# B&R Automation Studio project BaR_Automation_Studio
Automation Studio 4.9

## Configuration Config_5APC2100

CPU 5APC2100.BY48-000, AutomationRuntime B4.83, Build 4.1.2, Safety 1.10, Vc V4.72.6

### IoMap.iom - 5APC2100_BY48_000/IoMap.iom
```iecst
VAR_CONFIG
	::RESET_SAFETY AT %QX."X20SLX842".BOOL101;
	::Global_VInRoS_Str.EX_600.Slave.Info.Active AT %IX."EX600_WEN__V1_1".ModuleOk;
	::T_EX600:C_USINT_To_BOOL_Arr_1.INPUT AT %IB."EX600_WEN__V1_1".Module_0_Input011;
	::T_EX600:C_USINT_To_BOOL_Arr_2.INPUT AT %IB."EX600_WEN__V1_1".Module_0_Input012;
	::T_EX600:C_BOOL_Arr_To_USINT_1.OUTPUT AT %QB."EX600_WEN__V1_1".Module_0_Output003;
	::SAFETY_ACTIVE AT %IX."X20SLX842".SafeDigitalInput03;
	::SAFETY_STATUS AT %IX."X20SLX842".BOOL001;
	::T_ROB_1:ABB_Library_Rob_1.Status.PLC.Module_OK AT %IX."BASIC_V1_2".ModuleOk;
	::T_ROB_1:ABB_Library_Rob_1.PROFINET_Mapping_IN.STATUS.INPUT AT %IB."BASIC_V1_2".Module001_Input_0;
	::T_ROB_1:ABB_Library_Rob_1.PROFINET_Mapping_IN.SYSTEM.INPUT AT %IB."BASIC_V1_2".Module001_Input_1;
	::T_ROB_1:ABB_Library_Rob_1.PROFINET_Mapping_IN.STATE_uID AT %IB."BASIC_V1_2".Module001_Input_2;
	::T_ROB_1:ABB_Library_Rob_1.PROFINET_Mapping_IN.STATE_mID AT %IB."BASIC_V1_2".Module001_Input_3;
	::T_ROB_1:ABB_Library_Rob_1.PROFINET_Mapping_IN.MOTION_TRAJECTORY_ID.INPUT[0] AT %IB."BASIC_V1_2".Module001_Input_4;
	::T_ROB_1:ABB_Library_Rob_1.PROFINET_Mapping_IN.MOTION_TRAJECTORY_ID.INPUT[1] AT %IB."BASIC_V1_2".Module001_Input_5;
	::T_ROB_1:ABB_Library_Rob_1.PROFINET_Mapping_IN.JOINT_POS[0].INPUT[0] AT %IB."BASIC_V1_2".Module001_Input_6;
	::T_ROB_1:ABB_Library_Rob_1.PROFINET_Mapping_IN.JOINT_POS[0].INPUT[1] AT %IB."BASIC_V1_2".Module001_Input_7;
	::T_ROB_1:ABB_Library_Rob_1.PROFINET_Mapping_IN.JOINT_POS[1].INPUT[0] AT %IB."BASIC_V1_2".Module001_Input_8;
	::T_ROB_1:ABB_Library_Rob_1.PROFINET_Mapping_IN.JOINT_POS[1].INPUT[1] AT %IB."BASIC_V1_2".Module001_Input_9;
	::T_ROB_1:ABB_Library_Rob_1.PROFINET_Mapping_IN.JOINT_POS[2].INPUT[0] AT %IB."BASIC_V1_2".Module001_Input_10;
	::T_ROB_1:ABB_Library_Rob_1.PROFINET_Mapping_IN.JOINT_POS[2].INPUT[1] AT %IB."BASIC_V1_2".Module001_Input_11;
	::T_ROB_1:ABB_Library_Rob_1.PROFINET_Mapping_IN.JOINT_POS[3].INPUT[0] AT %IB."BASIC_V1_2".Module001_Input_12;
	::T_ROB_1:ABB_Library_Rob_1.PROFINET_Mapping_IN.JOINT_POS[3].INPUT[1] AT %IB."BASIC_V1_2".Module001_Input_13;
	::T_ROB_1:ABB_Library_Rob_1.PROFINET_Mapping_IN.JOINT_POS[4].INPUT[0] AT %IB."BASIC_V1_2".Module001_Input_14;
	::T_ROB_1:ABB_Library_Rob_1.PROFINET_Mapping_IN.JOINT_POS[4].INPUT[1] AT %IB."BASIC_V1_2".Module001_Input_15;
	::T_ROB_1:ABB_Library_Rob_1.PROFINET_Mapping_IN.JOINT_POS[5].INPUT[0] AT %IB."BASIC_V1_2".Module001_Input_16;
	::T_ROB_1:ABB_Library_Rob_1.PROFINET_Mapping_IN.JOINT_POS[5].INPUT[1] AT %IB."BASIC_V1_2".Module001_Input_17;
	::T_ROB_1:ABB_Library_Rob_1.PROFINET_Mapping_IN.JOINT_POS[6].INPUT[0] AT %IB."BASIC_V1_2".Module001_Input_18;
	::T_ROB_1:ABB_Library_Rob_1.PROFINET_Mapping_IN.JOINT_POS[6].INPUT[1] AT %IB."BASIC_V1_2".Module001_Input_19;
	::T_ROB_1:ABB_Library_Rob_1.PROFINET_Mapping_IN.JOINT_POS_SIGN.INPUT AT %IB."BASIC_V1_2".Module001_Input_20;
	::T_ROB_1:ABB_Library_Rob_1.PROFINET_Mapping_IN.TCP_POS[0].INPUT[0] AT %IB."BASIC_V1_2".Module001_Input_21;
	::T_ROB_1:ABB_Library_Rob_1.PROFINET_Mapping_IN.TCP_POS[0].INPUT[1] AT %IB."BASIC_V1_2".Module001_Input_22;
	::T_ROB_1:ABB_Library_Rob_1.PROFINET_Mapping_IN.TCP_POS[0].INPUT[2] AT %IB."BASIC_V1_2".Module001_Input_23;
	::T_ROB_1:ABB_Library_Rob_1.PROFINET_Mapping_IN.TCP_POS[0].INPUT[3] AT %IB."BASIC_V1_2".Module001_Input_24;
	::T_ROB_1:ABB_Library_Rob_1.PROFINET_Mapping_IN.TCP_POS[1].INPUT[0] AT %IB."BASIC_V1_2".Module001_Input_25;
	::T_ROB_1:ABB_Library_Rob_1.PROFINET_Mapping_IN.TCP_POS[1].INPUT[1] AT %IB."BASIC_V1_2".Module001_Input_26;
	::T_ROB_1:ABB_Library_Rob_1.PROFINET_Mapping_IN.TCP_POS[1].INPUT[2] AT %IB."BASIC_V1_2".Module001_Input_27;
	::T_ROB_1:ABB_Library_Rob_1.PROFINET_Mapping_IN.TCP_POS[1].INPUT[3] AT %IB."BASIC_V1_2".Module001_Input_28;
	::T_ROB_1:ABB_Library_Rob_1.PROFINET_Mapping_IN.TCP_POS[2].INPUT[0] AT %IB."BASIC_V1_2".Module001_Input_29;
	::T_ROB_1:ABB_Library_Rob_1.PROFINET_Mapping_IN.TCP_POS[2].INPUT[1] AT %IB."BASIC_V1_2".Module001_Input_30;
	::T_ROB_1:ABB_Library_Rob_1.PROFINET_Mapping_IN.TCP_POS[2].INPUT[2] AT %IB."BASIC_V1_2".Module001_Input_31;
	::T_ROB_1:ABB_Library_Rob_1.PROFINET_Mapping_IN.TCP_POS[2].INPUT[3] AT %IB."BASIC_V1_2".Module001_Input_32;
	::T_ROB_1:ABB_Library_Rob_1.PROFINET_Mapping_IN.TCP_ROT[0].INPUT[0] AT %IB."BASIC_V1_2".Module001_Input_33;
	::T_ROB_1:ABB_Library_Rob_1.PROFINET_Mapping_IN.TCP_ROT[0].INPUT[1] AT %IB."BASIC_V1_2".Module001_Input_34;
	::T_ROB_1:ABB_Library_Rob_1.PROFINET_Mapping_IN.TCP_ROT[1].INPUT[0] AT %IB."BASIC_V1_2".Module001_Input_35;
	::T_ROB_1:ABB_Library_Rob_1.PROFINET_Mapping_IN.TCP_ROT[1].INPUT[1] AT %IB."BASIC_V1_2".Module001_Input_36;
	::T_ROB_1:ABB_Library_Rob_1.PROFINET_Mapping_IN.TCP_ROT[2].INPUT[0] AT %IB."BASIC_V1_2".Module001_Input_37;
	::T_ROB_1:ABB_Library_Rob_1.PROFINET_Mapping_IN.TCP_ROT[2].INPUT[1] AT %IB."BASIC_V1_2".Module001_Input_38;
	::T_ROB_1:ABB_Library_Rob_1.PROFINET_Mapping_IN.TCP_EX_POS.INPUT[0] AT %IB."BASIC_V1_2".Module001_Input_39;
	::T_ROB_1:ABB_Library_Rob_1.PROFINET_Mapping_IN.TCP_EX_POS.INPUT[1] AT %IB."BASIC_V1_2".Module001_Input_40;
	::T_ROB_1:ABB_Library_Rob_1.PROFINET_Mapping_IN.TCP_SIGN.INPUT AT %IB."BASIC_V1_2".Module001_Input_41;
	::T_ROB_1:ABB_Library_Rob_1.PROFINET_Mapping_IN.TCP_CFG[0] AT %IB."BASIC_V1_2".Module001_Input_42;
	::T_ROB_1:ABB_Library_Rob_1.PROFINET_Mapping_IN.TCP_CFG[1] AT %IB."BASIC_V1_2".Module001_Input_43;
	::T_ROB_1:ABB_Library_Rob_1.PROFINET_Mapping_IN.TCP_CFG[2] AT %IB."BASIC_V1_2".Module001_Input_44;
	::T_ROB_1:ABB_Library_Rob_1.PROFINET_Mapping_IN.TCP_CFG[3] AT %IB."BASIC_V1_2".Module001_Input_45;
	::T_ROB_1:ABB_Library_Rob_1.PROFINET_Mapping_IN.TCP_CFG_SIGN.INPUT AT %IB."BASIC_V1_2".Module001_Input_46;
	::T_ROB_1:ABB_Library_Rob_1.PROFINET_Mapping_OUT.STATUS.OUTPUT AT %QB."BASIC_V1_2".Module002_Output_0;
	::T_ROB_1:ABB_Library_Rob_1.PROFINET_Mapping_OUT.SYSTEM.OUTPUT AT %QB."BASIC_V1_2".Module002_Output_1;
	::T_ROB_1:ABB_Library_Rob_1.PROFINET_Mapping_OUT.COMMAND.OUTPUT AT %QB."BASIC_V1_2".Module002_Output_2;
	::T_ROB_1:ABB_Library_Rob_1.PROFINET_Mapping_OUT.COMMAND_mID AT %QB."BASIC_V1_2".Module002_Output_3;
	::T_ROB_1:ABB_Library_Rob_1.PROFINET_Mapping_OUT.COMMAND_uID AT %QB."BASIC_V1_2".Module002_Output_4;
	::T_ROB_1:ABB_Library_Rob_1.PROFINET_Mapping_OUT.TRAJECTORY_SIZE.OUTPUT[0] AT %QB."BASIC_V1_2".Module002_Output_5;
	::T_ROB_1:ABB_Library_Rob_1.PROFINET_Mapping_OUT.TRAJECTORY_SIZE.OUTPUT[1] AT %QB."BASIC_V1_2".Module002_Output_6;
	::T_ROB_1:ABB_Library_Rob_1.PROFINET_Mapping_OUT.SPEED AT %QB."BASIC_V1_2".Module002_Output_7;
	::T_ROB_1:ABB_Library_Rob_1.PROFINET_Mapping_OUT.ZONE AT %QB."BASIC_V1_2".Module002_Output_8;
	::T_ROB_1:ABB_Library_Rob_1.PROFINET_Mapping_OUT.JOINT_POS[0].OUTPUT[0] AT %QB."BASIC_V1_2".Module002_Output_9;
	::T_ROB_1:ABB_Library_Rob_1.PROFINET_Mapping_OUT.JOINT_POS[0].OUTPUT[1] AT %QB."BASIC_V1_2".Module002_Output_10;
	::T_ROB_1:ABB_Library_Rob_1.PROFINET_Mapping_OUT.JOINT_POS[1].OUTPUT[0] AT %QB."BASIC_V1_2".Module002_Output_11;
	::T_ROB_1:ABB_Library_Rob_1.PROFINET_Mapping_OUT.JOINT_POS[1].OUTPUT[1] AT %QB."BASIC_V1_2".Module002_Output_12;
	::T_ROB_1:ABB_Library_Rob_1.PROFINET_Mapping_OUT.JOINT_POS[2].OUTPUT[0] AT %QB."BASIC_V1_2".Module002_Output_13;
	::T_ROB_1:ABB_Library_Rob_1.PROFINET_Mapping_OUT.JOINT_POS[2].OUTPUT[1] AT %QB."BASIC_V1_2".Module002_Output_14;
	::T_ROB_1:ABB_Library_Rob_1.PROFINET_Mapping_OUT.JOINT_POS[3].OUTPUT[0] AT %QB."BASIC_V1_2".Module002_Output_15;
	::T_ROB_1:ABB_Library_Rob_1.PROFINET_Mapping_OUT.JOINT_POS[3].OUTPUT[1] AT %QB."BASIC_V1_2".Module002_Output_16;
	::T_ROB_1:ABB_Library_Rob_1.PROFINET_Mapping_OUT.JOINT_POS[4].OUTPUT[0] AT %QB."BASIC_V1_2".Module002_Output_17;
	::T_ROB_1:ABB_Library_Rob_1.PROFINET_Mapping_OUT.JOINT_POS[4].OUTPUT[1] AT %QB."BASIC_V1_2".Module002_Output_18;
	::T_ROB_1:ABB_Library_Rob_1.PROFINET_Mapping_OUT.JOINT_POS[5].OUTPUT[0] AT %QB."BASIC_V1_2".Module002_Output_19;
	::T_ROB_1:ABB_Library_Rob_1.PROFINET_Mapping_OUT.JOINT_POS[5].OUTPUT[1] AT %QB."BASIC_V1_2".Module002_Output_20;
	::T_ROB_1:ABB_Library_Rob_1.PROFINET_Mapping_OUT.JOINT_POS[6].OUTPUT[0] AT %QB."BASIC_V1_2".Module002_Output_21;
	::T_ROB_1:ABB_Library_Rob_1.PROFINET_Mapping_OUT.JOINT_POS[6].OUTPUT[1] AT %QB."BASIC_V1_2".Module002_Output_22;
	::T_ROB_1:ABB_Library_Rob_1.PROFINET_Mapping_OUT.JOINT_POS_SIGN.OUTPUT AT %QB."BASIC_V1_2".Module002_Output_23;
	::T_ROB_1:ABB_Library_Rob_1.PROFINET_Mapping_OUT.TCP_POS[0].OUTPUT[0] AT %QB."BASIC_V1_2".Module002_Output_24;
	::T_ROB_1:ABB_Library_Rob_1.PROFINET_Mapping_OUT.TCP_POS[0].OUTPUT[1] AT %QB."BASIC_V1_2".Module002_Output_25;
	::T_ROB_1:ABB_Library_Rob_1.PROFINET_Mapping_OUT.TCP_POS[0].OUTPUT[2] AT %QB."BASIC_V1_2".Module002_Output_26;
	::T_ROB_1:ABB_Library_Rob_1.PROFINET_Mapping_OUT.TCP_POS[0].OUTPUT[3] AT %QB."BASIC_V1_2".Module002_Output_27;
	::T_ROB_1:ABB_Library_Rob_1.PROFINET_Mapping_OUT.TCP_POS[1].OUTPUT[0] AT %QB."BASIC_V1_2".Module002_Output_28;
	::T_ROB_1:ABB_Library_Rob_1.PROFINET_Mapping_OUT.TCP_POS[1].OUTPUT[1] AT %QB."BASIC_V1_2".Module002_Output_29;
	::T_ROB_1:ABB_Library_Rob_1.PROFINET_Mapping_OUT.TCP_POS[1].OUTPUT[2] AT %QB."BASIC_V1_2".Module002_Output_30;
	::T_ROB_1:ABB_Library_Rob_1.PROFINET_Mapping_OUT.TCP_POS[1].OUTPUT[3] AT %QB."BASIC_V1_2".Module002_Output_31;
	::T_ROB_1:ABB_Library_Rob_1.PROFINET_Mapping_OUT.TCP_POS[2].OUTPUT[0] AT %QB."BASIC_V1_2".Module002_Output_32;
	::T_ROB_1:ABB_Library_Rob_1.PROFINET_Mapping_OUT.TCP_POS[2].OUTPUT[1] AT %QB."BASIC_V1_2".Module002_Output_33;
	::T_ROB_1:ABB_Library_Rob_1.PROFINET_Mapping_OUT.TCP_POS[2].OUTPUT[2] AT %QB."BASIC_V1_2".Module002_Output_34;
	::T_ROB_1:ABB_Library_Rob_1.PROFINET_Mapping_OUT.TCP_POS[2].OUTPUT[3] AT %QB."BASIC_V1_2".Module002_Output_35;
	::T_ROB_1:ABB_Library_Rob_1.PROFINET_Mapping_OUT.TCP_ROT[0].OUTPUT[0] AT %QB."BASIC_V1_2".Module002_Output_36;
	::T_ROB_1:ABB_Library_Rob_1.PROFINET_Mapping_OUT.TCP_ROT[0].OUTPUT[1] AT %QB."BASIC_V1_2".Module002_Output_37;
	::T_ROB_1:ABB_Library_Rob_1.PROFINET_Mapping_OUT.TCP_ROT[1].OUTPUT[0] AT %QB."BASIC_V1_2".Module002_Output_38;
	::T_ROB_1:ABB_Library_Rob_1.PROFINET_Mapping_OUT.TCP_ROT[1].OUTPUT[1] AT %QB."BASIC_V1_2".Module002_Output_39;
	::T_ROB_1:ABB_Library_Rob_1.PROFINET_Mapping_OUT.TCP_ROT[2].OUTPUT[0] AT %QB."BASIC_V1_2".Module002_Output_40;
	::T_ROB_1:ABB_Library_Rob_1.PROFINET_Mapping_OUT.TCP_ROT[2].OUTPUT[1] AT %QB."BASIC_V1_2".Module002_Output_41;
	::T_ROB_1:ABB_Library_Rob_1.PROFINET_Mapping_OUT.TCP_EX_POS.OUTPUT[0] AT %QB."BASIC_V1_2".Module002_Output_42;
	::T_ROB_1:ABB_Library_Rob_1.PROFINET_Mapping_OUT.TCP_EX_POS.OUTPUT[1] AT %QB."BASIC_V1_2".Module002_Output_43;
	::T_ROB_1:ABB_Library_Rob_1.PROFINET_Mapping_OUT.TCP_SIGN.OUTPUT AT %QB."BASIC_V1_2".Module002_Output_44;
	::T_ROB_1:ABB_Library_Rob_1.PROFINET_Mapping_OUT.TCP_CFG[0] AT %QB."BASIC_V1_2".Module002_Output_45;
	::T_ROB_1:ABB_Library_Rob_1.PROFINET_Mapping_OUT.TCP_CFG[1] AT %QB."BASIC_V1_2".Module002_Output_46;
	::T_ROB_1:ABB_Library_Rob_1.PROFINET_Mapping_OUT.TCP_CFG[2] AT %QB."BASIC_V1_2".Module002_Output_47;
	::T_ROB_1:ABB_Library_Rob_1.PROFINET_Mapping_OUT.TCP_CFG[3] AT %QB."BASIC_V1_2".Module002_Output_48;
	::T_ROB_1:ABB_Library_Rob_1.PROFINET_Mapping_OUT.TCP_CFG_SIGN.OUTPUT AT %QB."BASIC_V1_2".Module002_Output_49;
	::T_ROB_1:ABB_Library_Rob_1.PROFINET_Mapping_OUT.RTOOL_RH.OUTPUT AT %QB."BASIC_V1_2".Module002_Output_50;
	::T_ROB_1:ABB_Library_Rob_1.PROFINET_Mapping_OUT.RTOOL_POS[0].OUTPUT[0] AT %QB."BASIC_V1_2".Module002_Output_51;
	::T_ROB_1:ABB_Library_Rob_1.PROFINET_Mapping_OUT.RTOOL_POS[0].OUTPUT[1] AT %QB."BASIC_V1_2".Module002_Output_52;
	::T_ROB_1:ABB_Library_Rob_1.PROFINET_Mapping_OUT.RTOOL_POS[1].OUTPUT[0] AT %QB."BASIC_V1_2".Module002_Output_53;
	::T_ROB_1:ABB_Library_Rob_1.PROFINET_Mapping_OUT.RTOOL_POS[1].OUTPUT[1] AT %QB."BASIC_V1_2".Module002_Output_54;
	::T_ROB_1:ABB_Library_Rob_1.PROFINET_Mapping_OUT.RTOOL_POS[2].OUTPUT[0] AT %QB."BASIC_V1_2".Module002_Output_55;
	::T_ROB_1:ABB_Library_Rob_1.PROFINET_Mapping_OUT.RTOOL_POS[2].OUTPUT[1] AT %QB."BASIC_V1_2".Module002_Output_56;
	::T_ROB_1:ABB_Library_Rob_1.PROFINET_Mapping_OUT.RTOOL_POS_SIGN.OUTPUT AT %QB."BASIC_V1_2".Module002_Output_57;
	::T_ROB_1:ABB_Library_Rob_1.PROFINET_Mapping_OUT.RTOOL_ROT_QUAT[0].OUTPUT[0] AT %QB."BASIC_V1_2".Module002_Output_58;
	::T_ROB_1:ABB_Library_Rob_1.PROFINET_Mapping_OUT.RTOOL_ROT_QUAT[0].OUTPUT[1] AT %QB."BASIC_V1_2".Module002_Output_59;
	::T_ROB_1:ABB_Library_Rob_1.PROFINET_Mapping_OUT.RTOOL_ROT_QUAT[0].OUTPUT[2] AT %QB."BASIC_V1_2".Module002_Output_60;
	::T_ROB_1:ABB_Library_Rob_1.PROFINET_Mapping_OUT.RTOOL_ROT_QUAT[0].OUTPUT[3] AT %QB."BASIC_V1_2".Module002_Output_61;
	::T_ROB_1:ABB_Library_Rob_1.PROFINET_Mapping_OUT.RTOOL_ROT_QUAT[1].OUTPUT[0] AT %QB."BASIC_V1_2".Module002_Output_62;
	::T_ROB_1:ABB_Library_Rob_1.PROFINET_Mapping_OUT.RTOOL_ROT_QUAT[1].OUTPUT[1] AT %QB."BASIC_V1_2".Module002_Output_63;
	::T_ROB_1:ABB_Library_Rob_1.PROFINET_Mapping_OUT.RTOOL_ROT_QUAT[1].OUTPUT[2] AT %QB."BASIC_V1_2".Module002_Output_64;
	::T_ROB_1:ABB_Library_Rob_1.PROFINET_Mapping_OUT.RTOOL_ROT_QUAT[1].OUTPUT[3] AT %QB."BASIC_V1_2".Module002_Output_65;
	::T_ROB_1:ABB_Library_Rob_1.PROFINET_Mapping_OUT.RTOOL_ROT_QUAT[2].OUTPUT[0] AT %QB."BASIC_V1_2".Module002_Output_66;
	::T_ROB_1:ABB_Library_Rob_1.PROFINET_Mapping_OUT.RTOOL_ROT_QUAT[2].OUTPUT[1] AT %QB."BASIC_V1_2".Module002_Output_67;
	::T_ROB_1:ABB_Library_Rob_1.PROFINET_Mapping_OUT.RTOOL_ROT_QUAT[2].OUTPUT[2] AT %QB."BASIC_V1_2".Module002_Output_68;
	::T_ROB_1:ABB_Library_Rob_1.PROFINET_Mapping_OUT.RTOOL_ROT_QUAT[2].OUTPUT[3] AT %QB."BASIC_V1_2".Module002_Output_69;
	::T_ROB_1:ABB_Library_Rob_1.PROFINET_Mapping_OUT.RTOOL_ROT_QUAT[3].OUTPUT[0] AT %QB."BASIC_V1_2".Module002_Output_70;
	::T_ROB_1:ABB_Library_Rob_1.PROFINET_Mapping_OUT.RTOOL_ROT_QUAT[3].OUTPUT[1] AT %QB."BASIC_V1_2".Module002_Output_71;
	::T_ROB_1:ABB_Library_Rob_1.PROFINET_Mapping_OUT.RTOOL_ROT_QUAT[3].OUTPUT[2] AT %QB."BASIC_V1_2".Module002_Output_72;
	::T_ROB_1:ABB_Library_Rob_1.PROFINET_Mapping_OUT.RTOOL_ROT_QUAT[3].OUTPUT[3] AT %QB."BASIC_V1_2".Module002_Output_73;
	::T_ROB_1:ABB_Library_Rob_1.PROFINET_Mapping_OUT.RTOOL_ROT_QUAT_SIGN.OUTPUT AT %QB."BASIC_V1_2".Module002_Output_74;
	::T_ROB_1:ABB_Library_Rob_1.PROFINET_Mapping_OUT.RTOOL_MASS.OUTPUT[0] AT %QB."BASIC_V1_2".Module002_Output_75;
	::T_ROB_1:ABB_Library_Rob_1.PROFINET_Mapping_OUT.RTOOL_MASS.OUTPUT[1] AT %QB."BASIC_V1_2".Module002_Output_76;
	::T_ROB_1:ABB_Library_Rob_1.PROFINET_Mapping_OUT.RTOOL_COG[0].OUTPUT[0] AT %QB."BASIC_V1_2".Module002_Output_77;
	::T_ROB_1:ABB_Library_Rob_1.PROFINET_Mapping_OUT.RTOOL_COG[0].OUTPUT[1] AT %QB."BASIC_V1_2".Module002_Output_78;
	::T_ROB_1:ABB_Library_Rob_1.PROFINET_Mapping_OUT.RTOOL_COG[0].OUTPUT[2] AT %QB."BASIC_V1_2".Module002_Output_79;
	::T_ROB_1:ABB_Library_Rob_1.PROFINET_Mapping_OUT.RTOOL_COG[0].OUTPUT[3] AT %QB."BASIC_V1_2".Module002_Output_80;
	::T_ROB_1:ABB_Library_Rob_1.PROFINET_Mapping_OUT.RTOOL_COG[1].OUTPUT[0] AT %QB."BASIC_V1_2".Module002_Output_81;
	::T_ROB_1:ABB_Library_Rob_1.PROFINET_Mapping_OUT.RTOOL_COG[1].OUTPUT[1] AT %QB."BASIC_V1_2".Module002_Output_82;
	::T_ROB_1:ABB_Library_Rob_1.PROFINET_Mapping_OUT.RTOOL_COG[1].OUTPUT[2] AT %QB."BASIC_V1_2".Module002_Output_83;
	::T_ROB_1:ABB_Library_Rob_1.PROFINET_Mapping_OUT.RTOOL_COG[1].OUTPUT[3] AT %QB."BASIC_V1_2".Module002_Output_84;
	::T_ROB_1:ABB_Library_Rob_1.PROFINET_Mapping_OUT.RTOOL_COG[2].OUTPUT[0] AT %QB."BASIC_V1_2".Module002_Output_85;
	::T_ROB_1:ABB_Library_Rob_1.PROFINET_Mapping_OUT.RTOOL_COG[2].OUTPUT[1] AT %QB."BASIC_V1_2".Module002_Output_86;
	::T_ROB_1:ABB_Library_Rob_1.PROFINET_Mapping_OUT.RTOOL_COG[2].OUTPUT[2] AT %QB."BASIC_V1_2".Module002_Output_87;
	::T_ROB_1:ABB_Library_Rob_1.PROFINET_Mapping_OUT.RTOOL_COG[2].OUTPUT[3] AT %QB."BASIC_V1_2".Module002_Output_88;
	::T_ROB_1:ABB_Library_Rob_1.PROFINET_Mapping_OUT.RTOOL_COG_SIGN.OUTPUT AT %QB."BASIC_V1_2".Module002_Output_89;
	::T_ROB_1:ABB_Library_Rob_1.PROFINET_Mapping_OUT.RTOOL_AOM_QUAT[0].OUTPUT[0] AT %QB."BASIC_V1_2".Module002_Output_90;
	::T_ROB_1:ABB_Library_Rob_1.PROFINET_Mapping_OUT.RTOOL_AOM_QUAT[0].OUTPUT[1] AT %QB."BASIC_V1_2".Module002_Output_91;
	::T_ROB_1:ABB_Library_Rob_1.PROFINET_Mapping_OUT.RTOOL_AOM_QUAT[0].OUTPUT[2] AT %QB."BASIC_V1_2".Module002_Output_92;
	::T_ROB_1:ABB_Library_Rob_1.PROFINET_Mapping_OUT.RTOOL_AOM_QUAT[0].OUTPUT[3] AT %QB."BASIC_V1_2".Module002_Output_93;
	::T_ROB_1:ABB_Library_Rob_1.PROFINET_Mapping_OUT.RTOOL_AOM_QUAT[1].OUTPUT[0] AT %QB."BASIC_V1_2".Module002_Output_94;
	::T_ROB_1:ABB_Library_Rob_1.PROFINET_Mapping_OUT.RTOOL_AOM_QUAT[1].OUTPUT[1] AT %QB."BASIC_V1_2".Module002_Output_95;
	::T_ROB_1:ABB_Library_Rob_1.PROFINET_Mapping_OUT.RTOOL_AOM_QUAT[1].OUTPUT[2] AT %QB."BASIC_V1_2".Module002_Output_96;
	::T_ROB_1:ABB_Library_Rob_1.PROFINET_Mapping_OUT.RTOOL_AOM_QUAT[1].OUTPUT[3] AT %QB."BASIC_V1_2".Module002_Output_97;
	::T_ROB_1:ABB_Library_Rob_1.PROFINET_Mapping_OUT.RTOOL_AOM_QUAT[2].OUTPUT[0] AT %QB."BASIC_V1_2".Module002_Output_98;
	::T_ROB_1:ABB_Library_Rob_1.PROFINET_Mapping_OUT.RTOOL_AOM_QUAT[2].OUTPUT[1] AT %QB."BASIC_V1_2".Module002_Output_99;
	::T_ROB_1:ABB_Library_Rob_1.PROFINET_Mapping_OUT.RTOOL_AOM_QUAT[2].OUTPUT[2] AT %QB."BASIC_V1_2".Module002_Output_100;
	::T_ROB_1:ABB_Library_Rob_1.PROFINET_Mapping_OUT.RTOOL_AOM_QUAT[2].OUTPUT[3] AT %QB."BASIC_V1_2".Module002_Output_101;
	::T_ROB_1:ABB_Library_Rob_1.PROFINET_Mapping_OUT.RTOOL_AOM_QUAT[3].OUTPUT[0] AT %QB."BASIC_V1_2".Module002_Output_102;
	::T_ROB_1:ABB_Library_Rob_1.PROFINET_Mapping_OUT.RTOOL_AOM_QUAT[3].OUTPUT[1] AT %QB."BASIC_V1_2".Module002_Output_103;
	::T_ROB_1:ABB_Library_Rob_1.PROFINET_Mapping_OUT.RTOOL_AOM_QUAT[3].OUTPUT[2] AT %QB."BASIC_V1_2".Module002_Output_104;
	::T_ROB_1:ABB_Library_Rob_1.PROFINET_Mapping_OUT.RTOOL_AOM_QUAT[3].OUTPUT[3] AT %QB."BASIC_V1_2".Module002_Output_105;
	::T_ROB_1:ABB_Library_Rob_1.PROFINET_Mapping_OUT.RTOOL_AOM_QUAT_SIGN.OUTPUT AT %QB."BASIC_V1_2".Module002_Output_106;
	::T_ROB_1:ABB_Library_Rob_1.PROFINET_Mapping_OUT.RTOOL_MOI[0].OUTPUT[0] AT %QB."BASIC_V1_2".Module002_Output_107;
	::T_ROB_1:ABB_Library_Rob_1.PROFINET_Mapping_OUT.RTOOL_MOI[0].OUTPUT[1] AT %QB."BASIC_V1_2".Module002_Output_108;
	::T_ROB_1:ABB_Library_Rob_1.PROFINET_Mapping_OUT.RTOOL_MOI[0].OUTPUT[2] AT %QB."BASIC_V1_2".Module002_Output_109;
	::T_ROB_1:ABB_Library_Rob_1.PROFINET_Mapping_OUT.RTOOL_MOI[0].OUTPUT[3] AT %QB."BASIC_V1_2".Module002_Output_110;
	::T_ROB_1:ABB_Library_Rob_1.PROFINET_Mapping_OUT.RTOOL_MOI[1].OUTPUT[0] AT %QB."BASIC_V1_2".Module002_Output_111;
	::T_ROB_1:ABB_Library_Rob_1.PROFINET_Mapping_OUT.RTOOL_MOI[1].OUTPUT[1] AT %QB."BASIC_V1_2".Module002_Output_112;
	::T_ROB_1:ABB_Library_Rob_1.PROFINET_Mapping_OUT.RTOOL_MOI[1].OUTPUT[2] AT %QB."BASIC_V1_2".Module002_Output_113;
	::T_ROB_1:ABB_Library_Rob_1.PROFINET_Mapping_OUT.RTOOL_MOI[1].OUTPUT[3] AT %QB."BASIC_V1_2".Module002_Output_114;
	::T_ROB_1:ABB_Library_Rob_1.PROFINET_Mapping_OUT.RTOOL_MOI[2].OUTPUT[0] AT %QB."BASIC_V1_2".Module002_Output_115;
	::T_ROB_1:ABB_Library_Rob_1.PROFINET_Mapping_OUT.RTOOL_MOI[2].OUTPUT[1] AT %QB."BASIC_V1_2".Module002_Output_116;
	::T_ROB_1:ABB_Library_Rob_1.PROFINET_Mapping_OUT.RTOOL_MOI[2].OUTPUT[2] AT %QB."BASIC_V1_2".Module002_Output_117;
	::T_ROB_1:ABB_Library_Rob_1.PROFINET_Mapping_OUT.RTOOL_MOI[2].OUTPUT[3] AT %QB."BASIC_V1_2".Module002_Output_118;
END_VAR
```

- Safety project (password-protected, skipped)

## Logical view

Binary libraries used (declarations not repeated): McAcpPar 5.22.2, McAxGroup

### Global.var
```iecst
VAR
	Global_VInRoS_Str : VInRoS_Str;
	RESET_SAFETY : BOOL;
	SAFETY_ACTIVE : BOOL;
	SAFETY_STATUS : BOOL;
	SIMULATION_ENABLE : BOOL;
	ROB_1_Sim_PROFINET_Mapping_OUT : ARRAY[0..255] OF USINT;
	ROB_1_Sim_PROFINET_Mapping_IN : ARRAY[0..255] OF USINT;
END_VAR
```

### Main.h
```c
#include <bur/plctypes.h>

#ifdef _DEFAULT_INCLUDES
	#include <AsDefault.h>
#endif

#define TRUE 1
#define FALSE (!TRUE)
#define NULL 0

typedef enum EX600_State_ID_enum{
	EX600_STATE_ACTIVE,
	EX600_STATE_HOME,
	EX600_STATE_WAIT,
	EX600_STATE_ERROR
}EX600_State_ID_enum;
```

### Program Logical/T_MECH_1

#### Main.c
```c
#include <bur/plctypes.h>

#ifdef _DEFAULT_INCLUDES
#include <AsDefault.h>
#endif

#include "Main.h"

_LOCAL struct MpAxisBasic MpAxisBasic_0;
_LOCAL struct MpAxisBasicParType AxisParameters;
_LOCAL enum Mechanism_State_ID_enum state_id;

void _INIT ProgramInit(void)
{
	memset(&Global_VInRoS_Str.Mech_Id_1, 0, sizeof(Global_VInRoS_Str.Mech_Id_1));

	AxisParameters.Homing.Mode = mcHOMING_ABSOLUTE;
	AxisParameters.Homing.Position = 1770365;

	MpAxisBasic_0.Enable     = 1;
	MpAxisBasic_0.MpLink     = &gAxis_Mech_01;
	MpAxisBasic_0.Parameters = &AxisParameters;

	Trajectory_Str.Targets.Position[0] = 100.0;
	Trajectory_Str.Targets.Position[1] = 1100.0;
	Trajectory_Str.Targets.Position[2] = 700.0;
	Trajectory_Str.Targets.Position[3] = 200.0;
	Trajectory_Str.Targets.Position[4] = 1200.0;

	Trajectory_Str.Targets.Velocity[0] = 500.0;
	Trajectory_Str.Targets.Velocity[1] = 1000.0;
	Trajectory_Str.Targets.Velocity[2] = 200.0;
	Trajectory_Str.Targets.Velocity[3] = 500.0;
	Trajectory_Str.Targets.Velocity[4] = 400.0;

	Trajectory_Str.Length = 5;

	state_id = MECH_STATE_ACTIVE;
}

void _CYCLIC ProgramCyclic(void)
{
	switch(state_id){
		case MECH_STATE_ACTIVE:
			{
				if(Global_VInRoS_Str.Mech_Id_1.Info.Active == TRUE){
					state_id = MECH_STATE_POWER;
				}
			}
			break;

		case MECH_STATE_POWER:
			{
				if(Global_VInRoS_Str.Mech_Id_1.Info.Power == TRUE){
					state_id = MECH_STATE_HOME;
				}
			}
			break;

		case MECH_STATE_HOME:
			{
				if(Global_VInRoS_Str.Mech_Id_1.Info.Home == TRUE){
					MpAxisBasic_0.Home = FALSE;
					Global_VInRoS_Str.Mech_Id_1.Command.Home = FALSE;
					state_id = MECH_STATE_WAIT;
				}
			}
			break;

		case MECH_STATE_WAIT:
			{
				if(Global_VInRoS_Str.Mech_Id_1.Command.Home == TRUE){
					state_id = MECH_STATE_HOME_UPD_PARAMETERS;
				}

				if(Global_VInRoS_Str.Mech_Id_1.Command.Start == TRUE){
					Trajectory_Str.Iteration = 0;
					state_id = MECH_STATE_UPD_PARAMETERS;
				}
			}
			break;

		case MECH_STATE_UPD_PARAMETERS:
			{
				Global_VInRoS_Str.Mech_Id_1.Parameters.Position = Trajectory_Str.Targets.Position[Trajectory_Str.Iteration];
				Global_VInRoS_Str.Mech_Id_1.Parameters.Velocity = Trajectory_Str.Targets.Velocity[Trajectory_Str.Iteration];
				Global_VInRoS_Str.Mech_Id_1.Parameters.Acc_Dec  = Trajectory_Str.Targets.Velocity[Trajectory_Str.Iteration]*10;

				Global_VInRoS_Str.Mech_Id_1.Command.Update = TRUE;
				if(Global_VInRoS_Str.Mech_Id_1.Info.Update_Done == TRUE){
					state_id = MECH_STATE_MOTION_1;
				}
			}
			break;

		case MECH_STATE_MOTION_1:
			{
				Global_VInRoS_Str.Mech_Id_1.Command.Move = TRUE;
				if(Global_VInRoS_Str.Mech_Id_1.Info.Move_Active == TRUE){
					state_id = MECH_STATE_MOTION_2;
				}
			}
			break;

		case MECH_STATE_MOTION_2:
			{
				if(Global_VInRoS_Str.Mech_Id_1.Command.Stop == TRUE){
					state_id = MECH_STATE_STOP;
				}else{
					if(Global_VInRoS_Str.Mech_Id_1.Info.In_Position == TRUE){
						Global_VInRoS_Str.Mech_Id_1.Command.Move = 0;

						if(Trajectory_Str.Iteration == Trajectory_Str.Length - 1){
							state_id = MECH_STATE_WAIT;
						}else{
							Trajectory_Str.Iteration++;
							state_id = MECH_STATE_UPD_PARAMETERS;
						}
					}
				}
			}
			break;

		case MECH_STATE_HOME_UPD_PARAMETERS:
			{
				Global_VInRoS_Str.Mech_Id_1.Parameters.Position = 700.0;
				Global_VInRoS_Str.Mech_Id_1.Parameters.Velocity = 500.0;
				Global_VInRoS_Str.Mech_Id_1.Parameters.Acc_Dec  = 5000.0;

				Global_VInRoS_Str.Mech_Id_1.Command.Update = TRUE;
				if(Global_VInRoS_Str.Mech_Id_1.Info.Update_Done == TRUE){
					state_id = MECH_STATE_HOME_MOTION_1;
				}
			}
			break;

		case MECH_STATE_HOME_MOTION_1:
			{
				Global_VInRoS_Str.Mech_Id_1.Command.Move = TRUE;
				if(Global_VInRoS_Str.Mech_Id_1.Info.Move_Active == TRUE){
					state_id = MECH_STATE_HOME_MOTION_2;
				}
			}
			break;

		case MECH_STATE_HOME_MOTION_2:
			{
				if(Global_VInRoS_Str.Mech_Id_1.Info.In_Position == TRUE){
					Global_VInRoS_Str.Mech_Id_1.Command.Move = FALSE;
					Global_VInRoS_Str.Mech_Id_1.Command.Home = FALSE;
					state_id = MECH_STATE_WAIT;
				}
			}
			break;

		case MECH_STATE_STOP:
			{
				Global_VInRoS_Str.Mech_Id_1.Command.Stop  = FALSE;
				Global_VInRoS_Str.Mech_Id_1.Command.Start = FALSE;

				Global_VInRoS_Str.Mech_Id_1.Command.Move = FALSE;
				if(Global_VInRoS_Str.Mech_Id_1.Info.Move_Active == FALSE){
					state_id = MECH_STATE_WAIT;
				}
			}
			break;

		case MECH_STATE_SAFETY:
			{
			}
			break;

		case MECH_STATE_ERROR:
			{
				Global_VInRoS_Str.Mech_Id_1.Command.Home   = FALSE;
				Global_VInRoS_Str.Mech_Id_1.Command.Update = FALSE;
				Global_VInRoS_Str.Mech_Id_1.Command.Stop   = FALSE;
				Global_VInRoS_Str.Mech_Id_1.Command.Start  = FALSE;
				Global_VInRoS_Str.Mech_Id_1.Command.Move   = FALSE;

				if(Global_VInRoS_Str.Mech_Id_1.Info.Error == FALSE){
					state_id = MECH_STATE_WAIT;
				}
			}
			break;

	}

	AxisParameters.Position     = Global_VInRoS_Str.Mech_Id_1.Parameters.Position;
	AxisParameters.Velocity     = Global_VInRoS_Str.Mech_Id_1.Parameters.Velocity;
	AxisParameters.Acceleration = Global_VInRoS_Str.Mech_Id_1.Parameters.Acc_Dec;
	AxisParameters.Deceleration = Global_VInRoS_Str.Mech_Id_1.Parameters.Acc_Dec;

	MpAxisBasic_0.Power = Global_VInRoS_Str.Mech_Id_1.Command.Power;
	if(Global_VInRoS_Str.Mech_Id_1.Command.Home == TRUE && Global_VInRoS_Str.Mech_Id_1.Info.Home == FALSE){
		MpAxisBasic_0.Home = TRUE;
	}
	MpAxisBasic_0.ErrorReset = Global_VInRoS_Str.Mech_Id_1.Command.Reset_Error;
	MpAxisBasic_0.Update     = Global_VInRoS_Str.Mech_Id_1.Command.Update;
	MpAxisBasic_0.MoveAbsolute = Global_VInRoS_Str.Mech_Id_1.Command.Move;

	MpAxisBasic(&MpAxisBasic_0);

	Global_VInRoS_Str.Mech_Id_1.Info.Active = MpAxisBasic_0.Active;
	Global_VInRoS_Str.Mech_Id_1.Info.Power  = MpAxisBasic_0.PowerOn;
	Global_VInRoS_Str.Mech_Id_1.Info.Home   = MpAxisBasic_0.IsHomed;
	Global_VInRoS_Str.Mech_Id_1.Info.Error  = MpAxisBasic_0.Error;
	Global_VInRoS_Str.Mech_Id_1.Info.Update_Done = MpAxisBasic_0.UpdateDone;
	Global_VInRoS_Str.Mech_Id_1.Info.Move_Active = MpAxisBasic_0.MoveActive;
	if(MpAxisBasic_0.InPosition == TRUE && MpAxisBasic_0.MoveDone == TRUE){
		Global_VInRoS_Str.Mech_Id_1.Info.In_Position = TRUE;
	}else{
		Global_VInRoS_Str.Mech_Id_1.Info.In_Position = FALSE;
	}
	Global_VInRoS_Str.Mech_Id_1.Info.Safety = FALSE;

	Global_VInRoS_Str.Mech_Id_1.Position = MpAxisBasic_0.Position;

	if(Global_VInRoS_Str.Mech_Id_1.Info.Error == TRUE){
		state_id = MECH_STATE_ERROR;
	}
}
```

### Types.typ
```iecst
TYPE
	Traj_Str : 	STRUCT
		Targets : Targets_Str;
		Length : USINT;
		Iteration : USINT;
	END_STRUCT;
	Targets_Str : 	STRUCT
		Position : ARRAY[0..99]OF LREAL;
		Velocity : ARRAY[0..99]OF REAL;
	END_STRUCT;
END_TYPE
```

### Variables.var
```iecst
VAR
	Trajectory_Str : Traj_Str;
END_VAR
```

### Program Logical/T_ROB_1

#### Main.c
```c
#include <bur/plctypes.h>

#ifdef _DEFAULT_INCLUDES
#include <AsDefault.h>
#endif

#include <Main.h>

_LOCAL enum Robot_State_ID_enum state_id;

void _INIT ProgramInit(void)
{
	//
	memset(&Global_VInRoS_Str.Rob_Id_1, 0, sizeof(Global_VInRoS_Str.Rob_Id_1));

	ABB_Library_Rob_1.Enable = TRUE;

	//
	ABB_Library_Rob_1.Rob_Tool.robHold = FALSE;
	ABB_Library_Rob_1.Rob_Tool.tFrame.Position[0] = 0.0; ABB_Library_Rob_1.Rob_Tool.tFrame.Position[1] = 0.0;
	ABB_Library_Rob_1.Rob_Tool.tFrame.Position[2] = 0.0;
	ABB_Library_Rob_1.Rob_Tool.tFrame.Rotation[0] = 1.0; ABB_Library_Rob_1.Rob_Tool.tFrame.Rotation[1] = 0.0;
	ABB_Library_Rob_1.Rob_Tool.tFrame.Rotation[2] = 0.0; ABB_Library_Rob_1.Rob_Tool.tFrame.Rotation[3] = 0.0;
	ABB_Library_Rob_1.Rob_Tool.tLoad.mass = 0.0;
	ABB_Library_Rob_1.Rob_Tool.tLoad.center_of_gravity[0] = 0.0; ABB_Library_Rob_1.Rob_Tool.tLoad.center_of_gravity[1] = 0.0;
	ABB_Library_Rob_1.Rob_Tool.tLoad.center_of_gravity[2] = 0.0;
	ABB_Library_Rob_1.Rob_Tool.tLoad.intertial_axes[0] = 1.0; ABB_Library_Rob_1.Rob_Tool.tLoad.intertial_axes[1] = 0.0;
	ABB_Library_Rob_1.Rob_Tool.tLoad.intertial_axes[2] = 0.0; ABB_Library_Rob_1.Rob_Tool.tLoad.intertial_axes[3] = 0.0;
	ABB_Library_Rob_1.Rob_Tool.tLoad.moment_of_inertia[0] = 0.0; ABB_Library_Rob_1.Rob_Tool.tLoad.moment_of_inertia[1] = 0.0;
	ABB_Library_Rob_1.Rob_Tool.tLoad.moment_of_inertia[2] = 0.0;

	//
	Set_Trajectory_Parameters(&Trajectory_Str);
}

void _CYCLIC ProgramCyclic(void)
{
	switch(state_id){
		case ROB_STATE_ACTIVE:
			{
				if(Global_VInRoS_Str.Rob_Id_1.Info.Active == TRUE){
					state_id = ROB_STATE_POWER;
				}
			}
			break;

		case ROB_STATE_POWER:
			{
				if(Global_VInRoS_Str.Rob_Id_1.Command.Power == TRUE){
					ABB_Library_Rob_1.Power_ON = TRUE;
					Global_VInRoS_Str.Rob_Id_1.Command.Power = FALSE;
				}

				if(Global_VInRoS_Str.Rob_Id_1.Info.Power == TRUE && ABB_Library_Rob_1.Status.Robot.ID.Motion == ABBr_STATE_WAIT){
					state_id = ROB_STATE_WAIT;
				}
			}
			break;

		case ROB_STATE_WAIT:
			{
				ABB_Library_Rob_1.Command.STOP  = FALSE;
				ABB_Library_Rob_1.Command.START = FALSE;

				if(Global_VInRoS_Str.Rob_Id_1.Command.Home == TRUE){
					state_id = ROB_STATE_HOME_UPD_PARAMETERS_1;
				}

				if(Global_VInRoS_Str.Rob_Id_1.Command.Start == TRUE){
					state_id = ROB_STATE_UPD_PARAMETERS_1;
				}
			}
			break;

		case ROB_STATE_UPD_PARAMETERS_1:
			{
				Global_VInRoS_Str.Rob_Id_1.Info.Update_Done = FALSE;

				memcpy(ABB_Library_Rob_1.Parameter.Joint, Trajectory_Str.Targets.Joint,
					(sizeof(Trajectory_Str.Targets.Joint) / sizeof(Trajectory_Str.Targets.Joint[0])) * sizeof(REAL));
				int i;
				for(i = 0; i < Trajectory_Str.Length; i++){
					ABB_Library_Rob_1.Parameter.Speed[i] = Trajectory_Str.Targets.Speed[i];
					ABB_Library_Rob_1.Parameter.Zone[i] = Trajectory_Str.Targets.Zone[i];
				}

				ABB_Library_Rob_1.Parameter.Trajectory_Size = Trajectory_Str.Length;

				ABB_Library_Rob_1.Command.ID.Update = UPT_ID_TRAJECTORY_JOINT;
				ABB_Library_Rob_1.Command.UPDATE    = TRUE;

				if(ABB_Library_Rob_1.Internal.Update.actual_state != UPT_STATE_WAIT){
					state_id = ROB_STATE_UPD_PARAMETERS_2;
				}
			}
			break;

		case ROB_STATE_UPD_PARAMETERS_2:
			{
				if(ABB_Library_Rob_1.Status.Robot.Update_Done == TRUE && ABB_Library_Rob_1.Internal.Update.actual_state == UPT_STATE_WAIT){
					Global_VInRoS_Str.Rob_Id_1.Info.Update_Done = TRUE;
					state_id = ROB_STATE_MOTION_1;
				}
			}
			break;

		case ROB_STATE_MOTION_1:
			{
				ABB_Library_Rob_1.Command.ID.Motion = MAIN_ID_JOINT_ABSOLUTE;
				ABB_Library_Rob_1.Command.START = TRUE;

				if(Global_VInRoS_Str.Rob_Id_1.Info.Move_Active == TRUE){
					state_id = ROB_STATE_MOTION_2;
				}
			}
			break;

		case ROB_STATE_MOTION_2:
			{
				ABB_Library_Rob_1.Command.START = FALSE;

				Trajectory_Str.Iteration = ABB_Library_Rob_1.Status.Robot.Trajectory_ID;

				if(Global_VInRoS_Str.Rob_Id_1.Command.Stop == TRUE){
					state_id = ROB_STATE_STOP;
				}else{
					if(Global_VInRoS_Str.Rob_Id_1.Info.In_Position == TRUE){
						state_id = ROB_STATE_WAIT;
					}
				}
			}
			break;

		case ROB_STATE_HOME_UPD_PARAMETERS_1:
			{
				Global_VInRoS_Str.Rob_Id_1.Info.Update_Done = FALSE;
				Global_VInRoS_Str.Rob_Id_1.Command.Home = FALSE;

				ABB_Library_Rob_1.Parameter.Joint[0].Q[0] = 90.0; ABB_Library_Rob_1.Parameter.Joint[0].Q[1] = 0.0;
				ABB_Library_Rob_1.Parameter.Joint[0].Q[2] = 0.0; ABB_Library_Rob_1.Parameter.Joint[0].Q[3] = 0.0;
				ABB_Library_Rob_1.Parameter.Joint[0].Q[4] = 90.0; ABB_Library_Rob_1.Parameter.Joint[0].Q[5] = 0.0;
				ABB_Library_Rob_1.Parameter.Speed[0] = vSPEED_100;
				ABB_Library_Rob_1.Parameter.Zone[0]  = zZone_fine;

				ABB_Library_Rob_1.Parameter.Trajectory_Size = 1;

				ABB_Library_Rob_1.Command.ID.Update = UPT_ID_TRAJECTORY_JOINT;
				ABB_Library_Rob_1.Command.UPDATE    = TRUE;

				if(ABB_Library_Rob_1.Internal.Update.actual_state != UPT_STATE_WAIT){
					state_id = ROB_STATE_HOME_UPD_PARAMETERS_2;
				}
			}
			break;

		case ROB_STATE_HOME_UPD_PARAMETERS_2:
			{
				if(ABB_Library_Rob_1.Status.Robot.Update_Done == TRUE && ABB_Library_Rob_1.Internal.Update.actual_state == UPT_STATE_WAIT){
					Global_VInRoS_Str.Rob_Id_1.Info.Update_Done = TRUE;
					state_id = ROB_STATE_HOME_MOTION_1;
				}
			}
			break;

		case ROB_STATE_HOME_MOTION_1:
			{
				Global_VInRoS_Str.Rob_Id_1.Info.Home = FALSE;

				ABB_Library_Rob_1.Command.ID.Motion = MAIN_ID_JOINT_ABSOLUTE;
				ABB_Library_Rob_1.Command.START = TRUE;

				if(Global_VInRoS_Str.Rob_Id_1.Info.Move_Active == TRUE){
					state_id = ROB_STATE_HOME_MOTION_2;
				}
			}
			break;

		case ROB_STATE_HOME_MOTION_2:
			{
				ABB_Library_Rob_1.Command.START = FALSE;

				if(Global_VInRoS_Str.Rob_Id_1.Command.Stop == TRUE){
					state_id = ROB_STATE_STOP;
				}else{
					if(Global_VInRoS_Str.Rob_Id_1.Info.In_Position == TRUE){
						Global_VInRoS_Str.Rob_Id_1.Info.Home = TRUE;
						state_id = ROB_STATE_WAIT;
					}
				}
			}
			break;

		case ROB_STATE_STOP:
			{
				Global_VInRoS_Str.Rob_Id_1.Command.Home  = FALSE;
				Global_VInRoS_Str.Rob_Id_1.Command.Start = FALSE;
				Global_VInRoS_Str.Rob_Id_1.Command.Stop  = FALSE;

				if(ABB_Library_Rob_1.Internal.actual_state == ABBt_STATE_WAIT && ABB_Library_Rob_1.Status.Robot.ID.Motion == ABBr_STATE_WAIT){
					state_id = ROB_STATE_WAIT;
				}else{
					ABB_Library_Rob_1.Command.STOP = TRUE;
				}
			}
			break;

		case ROB_STATE_SAFETY:
			{
			}
			break;

		case ROB_STATE_ERROR:
			{
			}
			break;
	}

	ABB_Library(&ABB_Library_Rob_1);

	Global_VInRoS_Str.Rob_Id_1.Info.Active = ABB_Library_Rob_1.Status.Robot.Active;
	Global_VInRoS_Str.Rob_Id_1.Info.Power = ABB_Library_Rob_1.Status.Robot.System.MOTOR_ON;
	if(ABB_Library_Rob_1.Status.Robot.In_Position == TRUE && ABB_Library_Rob_1.Status.Robot.ID.Motion == ABBr_STATE_WAIT){
		Global_VInRoS_Str.Rob_Id_1.Info.In_Position = TRUE;
	}else{
		Global_VInRoS_Str.Rob_Id_1.Info.In_Position = FALSE;
	}
	Global_VInRoS_Str.Rob_Id_1.Info.Error  = FALSE;
	Global_VInRoS_Str.Rob_Id_1.Info.Safety = FALSE;

	if(Global_VInRoS_Str.Rob_Id_1.Info.Power == TRUE){
		if(Global_VInRoS_Str.Rob_Id_1.Info.In_Position == FALSE){
			Global_VInRoS_Str.Rob_Id_1.Info.Move_Active = TRUE;
		}else{
			Global_VInRoS_Str.Rob_Id_1.Info.Move_Active = FALSE;
		}
	}

	memcpy(Global_VInRoS_Str.Rob_Id_1.Position.Q, ABB_Library_Rob_1.RT_Data.Q,
		(sizeof(ABB_Library_Rob_1.RT_Data.Q) / sizeof(ABB_Library_Rob_1.RT_Data.Q[0])) * sizeof(REAL));

	if(Global_VInRoS_Str.Rob_Id_1.Info.Error == TRUE){
		state_id = ROB_STATE_ERROR;
	}
}
```

### Program Logical/T_ROB_2_L (ANSIC)

#### Main.c - Init, cyclic, exit code
```c
#include <bur/plctypes.h>

#ifdef _DEFAULT_INCLUDES
#include <AsDefault.h>
#endif

#include <Main.h>

_LOCAL enum Robot_State_ID_enum state_id;

void _INIT ProgramInit(void)
{
	//
	memset(&Global_VInRoS_Str.Rob_Id_2_L, 0, sizeof(Global_VInRoS_Str.Rob_Id_2_L));

	ABB_Library_Rob_1.Enable = TRUE;

	//
	ABB_Library_Rob_1.Rob_Tool.robHold = FALSE;
	ABB_Library_Rob_1.Rob_Tool.tFrame.Position[0] = 0.0; ABB_Library_Rob_1.Rob_Tool.tFrame.Position[1] = 0.0;
	ABB_Library_Rob_1.Rob_Tool.tFrame.Position[2] = 0.0;
	ABB_Library_Rob_1.Rob_Tool.tFrame.Rotation[0] = 1.0; ABB_Library_Rob_1.Rob_Tool.tFrame.Rotation[1] = 0.0;
	ABB_Library_Rob_1.Rob_Tool.tFrame.Rotation[2] = 0.0; ABB_Library_Rob_1.Rob_Tool.tFrame.Rotation[3] = 0.0;
	ABB_Library_Rob_1.Rob_Tool.tLoad.mass = 0.0;
	ABB_Library_Rob_1.Rob_Tool.tLoad.center_of_gravity[0] = 0.0; ABB_Library_Rob_1.Rob_Tool.tLoad.center_of_gravity[1] = 0.0;
	ABB_Library_Rob_1.Rob_Tool.tLoad.center_of_gravity[2] = 0.0;
	ABB_Library_Rob_1.Rob_Tool.tLoad.intertial_axes[0] = 1.0; ABB_Library_Rob_1.Rob_Tool.tLoad.intertial_axes[1] = 0.0;
	ABB_Library_Rob_1.Rob_Tool.tLoad.intertial_axes[2] = 0.0; ABB_Library_Rob_1.Rob_Tool.tLoad.intertial_axes[3] = 0.0;
	ABB_Library_Rob_1.Rob_Tool.tLoad.moment_of_inertia[0] = 0.0; ABB_Library_Rob_1.Rob_Tool.tLoad.moment_of_inertia[1] = 0.0;
	ABB_Library_Rob_1.Rob_Tool.tLoad.moment_of_inertia[2] = 0.0;

	//
	Set_Trajectory_Parameters(&Trajectory_Str, 30.0);
}

void _CYCLIC ProgramCyclic(void)
{
	switch(state_id){
		case ROB_STATE_ACTIVE:
			{
				if(Global_VInRoS_Str.Rob_Id_2_L.Info.Active == TRUE){
					state_id = ROB_STATE_POWER;
				}
			}
			break;

		case ROB_STATE_POWER:
			{
				if(Global_VInRoS_Str.Rob_Id_2_L.Command.Power == TRUE){
					ABB_Library_Rob_1.Power_ON = TRUE;
					Global_VInRoS_Str.Rob_Id_2_L.Command.Power = FALSE;
				}

				if(Global_VInRoS_Str.Rob_Id_2_L.Info.Power == TRUE && ABB_Library_Rob_1.Status.Robot.ID.Motion == ABBr_STATE_WAIT){
					state_id = ROB_STATE_WAIT;
				}
			}
			break;

		case ROB_STATE_WAIT:
			{
				ABB_Library_Rob_1.Command.STOP  = FALSE;
				ABB_Library_Rob_1.Command.START = FALSE;

				if(Global_VInRoS_Str.Rob_Id_2_L.Command.Home == TRUE){
					state_id = ROB_STATE_HOME_UPD_PARAMETERS_1;
				}

				if(Global_VInRoS_Str.Rob_Id_2_L.Command.Start == TRUE){
					state_id = ROB_STATE_UPD_PARAMETERS_1;
				}
			}
			break;

		case ROB_STATE_UPD_PARAMETERS_1:
			{
				Global_VInRoS_Str.Rob_Id_2_L.Info.Update_Done = FALSE;

				memcpy(ABB_Library_Rob_1.Parameter.Joint, Trajectory_Str.Targets.Joint,
					(sizeof(Trajectory_Str.Targets.Joint) / sizeof(Trajectory_Str.Targets.Joint[0])) * sizeof(REAL));
				int i;
				for(i = 0; i < Trajectory_Str.Length; i++){
					ABB_Library_Rob_1.Parameter.Speed[i] = Trajectory_Str.Targets.Speed[i];
					ABB_Library_Rob_1.Parameter.Zone[i] = Trajectory_Str.Targets.Zone[i];
				}

				ABB_Library_Rob_1.Parameter.Trajectory_Size = Trajectory_Str.Length;

				ABB_Library_Rob_1.Command.ID.Update = UPT_ID_TRAJECTORY_JOINT;
				ABB_Library_Rob_1.Command.UPDATE    = TRUE;

				if(ABB_Library_Rob_1.Internal.Update.actual_state != UPT_STATE_WAIT){
					state_id = ROB_STATE_UPD_PARAMETERS_2;
				}
			}
			break;

		case ROB_STATE_UPD_PARAMETERS_2:
			{
				if(ABB_Library_Rob_1.Status.Robot.Update_Done == TRUE && ABB_Library_Rob_1.Internal.Update.actual_state == UPT_STATE_WAIT){
					Global_VInRoS_Str.Rob_Id_2_L.Info.Update_Done = TRUE;
					state_id = ROB_STATE_MOTION_1;
				}
			}
			break;

		case ROB_STATE_MOTION_1:
			{
				ABB_Library_Rob_1.Command.ID.Motion = MAIN_ID_JOINT_ABSOLUTE;
				ABB_Library_Rob_1.Command.START = TRUE;

				if(Global_VInRoS_Str.Rob_Id_2_L.Info.Move_Active == TRUE){
					state_id = ROB_STATE_MOTION_2;
				}
			}
			break;

		case ROB_STATE_MOTION_2:
			{
				ABB_Library_Rob_1.Command.START = FALSE;

				Trajectory_Str.Iteration = ABB_Library_Rob_1.Status.Robot.Trajectory_ID;

				if(Global_VInRoS_Str.Rob_Id_2_L.Command.Stop == TRUE){
					state_id = ROB_STATE_STOP;
				}else{
					if(Global_VInRoS_Str.Rob_Id_2_L.Info.In_Position == TRUE){
						state_id = ROB_STATE_WAIT;
					}
				}
			}
			break;

		case ROB_STATE_HOME_UPD_PARAMETERS_1:
			{
				Global_VInRoS_Str.Rob_Id_2_L.Info.Update_Done = FALSE;
				Global_VInRoS_Str.Rob_Id_2_L.Command.Home = FALSE;

				ABB_Library_Rob_1.Parameter.Joint[0].Q[0] = 0.0; ABB_Library_Rob_1.Parameter.Joint[0].Q[1] = -130.0;
				ABB_Library_Rob_1.Parameter.Joint[0].Q[2] = 30.0; ABB_Library_Rob_1.Parameter.Joint[0].Q[3] = 0.0;
				ABB_Library_Rob_1.Parameter.Joint[0].Q[4] = 40.0; ABB_Library_Rob_1.Parameter.Joint[0].Q[5] = 0.0;
				ABB_Library_Rob_1.Parameter.Joint[0].Q[6] = 135.0;
				ABB_Library_Rob_1.Parameter.Speed[0] = vSPEED_100;
				ABB_Library_Rob_1.Parameter.Zone[0]  = zZone_fine;

				ABB_Library_Rob_1.Parameter.Trajectory_Size = 1;

				ABB_Library_Rob_1.Command.ID.Update = UPT_ID_TRAJECTORY_JOINT;
				ABB_Library_Rob_1.Command.UPDATE    = TRUE;

				if(ABB_Library_Rob_1.Internal.Update.actual_state != UPT_STATE_WAIT){
					state_id = ROB_STATE_HOME_UPD_PARAMETERS_2;
				}
			}
			break;

		case ROB_STATE_HOME_UPD_PARAMETERS_2:
			{
				if(ABB_Library_Rob_1.Status.Robot.Update_Done == TRUE && ABB_Library_Rob_1.Internal.Update.actual_state == UPT_STATE_WAIT){
					Global_VInRoS_Str.Rob_Id_2_L.Info.Update_Done = TRUE;
					state_id = ROB_STATE_HOME_MOTION_1;
				}
			}
			break;

		case ROB_STATE_HOME_MOTION_1:
			{
				Global_VInRoS_Str.Rob_Id_2_L.Info.Home = FALSE;

				ABB_Library_Rob_1.Command.ID.Motion = MAIN_ID_JOINT_ABSOLUTE;
				ABB_Library_Rob_1.Command.START = TRUE;

				if(Global_VInRoS_Str.Rob_Id_2_L.Info.Move_Active == TRUE){
					state_id = ROB_STATE_HOME_MOTION_2;
				}
			}
			break;

		case ROB_STATE_HOME_MOTION_2:
			{
				ABB_Library_Rob_1.Command.START = FALSE;

				if(Global_VInRoS_Str.Rob_Id_2_L.Command.Stop == TRUE){
					state_id = ROB_STATE_STOP;
				}else{
					if(Global_VInRoS_Str.Rob_Id_2_L.Info.In_Position == TRUE){
						Global_VInRoS_Str.Rob_Id_2_L.Info.Home = TRUE;
						state_id = ROB_STATE_WAIT;
					}
				}
			}
			break;

		case ROB_STATE_STOP:
			{
				Global_VInRoS_Str.Rob_Id_2_L.Command.Home  = FALSE;
				Global_VInRoS_Str.Rob_Id_2_L.Command.Start = FALSE;
				Global_VInRoS_Str.Rob_Id_2_L.Command.Stop  = FALSE;

				if(ABB_Library_Rob_1.Internal.actual_state == ABBt_STATE_WAIT && ABB_Library_Rob_1.Status.Robot.ID.Motion == ABBr_STATE_WAIT){
					state_id = ROB_STATE_WAIT;
				}else{
					ABB_Library_Rob_1.Command.STOP = TRUE;
				}
			}
			break;

		case ROB_STATE_SAFETY:
			{
			}
			break;

		case ROB_STATE_ERROR:
			{
			}
			break;
	}

	ABB_Library(&ABB_Library_Rob_1);

	Global_VInRoS_Str.Rob_Id_2_L.Info.Active = ABB_Library_Rob_1.Status.Robot.Active;
	Global_VInRoS_Str.Rob_Id_2_L.Info.Power = ABB_Library_Rob_1.Status.Robot.System.MOTOR_ON;
	if(ABB_Library_Rob_1.Status.Robot.In_Position == TRUE && ABB_Library_Rob_1.Status.Robot.ID.Motion == ABBr_STATE_WAIT){
		Global_VInRoS_Str.Rob_Id_2_L.Info.In_Position = TRUE;
	}else{
		Global_VInRoS_Str.Rob_Id_2_L.Info.In_Position = FALSE;
	}
	Global_VInRoS_Str.Rob_Id_2_L.Info.Error  = FALSE;
	Global_VInRoS_Str.Rob_Id_2_L.Info.Safety = FALSE;

	if(Global_VInRoS_Str.Rob_Id_2_L.Info.Power == TRUE){
		if(Global_VInRoS_Str.Rob_Id_2_L.Info.In_Position == FALSE){
			Global_VInRoS_Str.Rob_Id_2_L.Info.Move_Active = TRUE;
		}else{
			Global_VInRoS_Str.Rob_Id_2_L.Info.Move_Active = FALSE;
		}
	}

	memcpy(Global_VInRoS_Str.Rob_Id_2_L.Position.Q, ABB_Library_Rob_1.RT_Data.Q,
		(sizeof(ABB_Library_Rob_1.RT_Data.Q) / sizeof(ABB_Library_Rob_1.RT_Data.Q[0])) * sizeof(REAL));

	if(Global_VInRoS_Str.Rob_Id_2_L.Info.Error == TRUE){
		state_id = ROB_STATE_ERROR;
	}
}
```

#### Types.typ
```iecst
TYPE
	Traj_Str : 	STRUCT
		Targets : Targets_Str;
		Length : USINT;
		Iteration : USINT;
	END_STRUCT;
	Targets_Str : 	STRUCT
		Joint : ARRAY[0..99]OF Targets_Joint_Str;
		Speed : ARRAY[0..99]OF USINT;
		Zone : ARRAY[0..99]OF USINT;
	END_STRUCT;
	Targets_Joint_Str : 	STRUCT
		Q : ARRAY[0..6]OF REAL;
	END_STRUCT;
END_TYPE
```

### Converter.h
```c
/**
 * MIT License
 * Copyright(c) 2022 Roman Parak
 * Permission is hereby granted, free of charge, to any person obtaining a copy
 * of this software and associated documentation files (the "Software"), to deal
 * in the Software without restriction, including without limitation the rights
 * to use, copy, modify, merge, publish, distribute, sublicense, and/or sell
 * copies of the Software, and to permit persons to whom the Software is
 * furnished to do so, subject to the following conditions:
 * The above copyright notice and this permission notice shall be included in all
 * copies or substantial portions of the Software.
 * THE SOFTWARE IS PROVIDED "AS IS", WITHOUT WARRANTY OF ANY KIND, EXPRESS OR
 * IMPLIED, INCLUDING BUT NOT LIMITED TO THE WARRANTIES OF MERCHANTABILITY,
 * FITNESS FOR A PARTICULAR PURPOSE AND NONINFRINGEMENT. IN NO EVENT SHALL THE
 * AUTHORS OR COPYRIGHT HOLDERS BE LIABLE FOR ANY CLAIM, DAMAGES OR OTHER
 * LIABILITY, WHETHER IN AN ACTION OF CONTRACT, TORT OR OTHERWISE, ARISING FROM,
 * OUT OF OR IN CONNECTION WITH THE SOFTWARE OR THE USE OR OTHER DEALINGS IN THE
 * SOFTWARE.
 */

/**
 * Author   : Roman Parak
 * Email    : Roman.Parak@outlook.com
 * File Name: Converter.h
 * Github   : https://github.com/rparak
 */

#ifndef HEADER_FILE_CONVERTER
#define HEADER_FILE_CONVERTER

/** < Include B&R Automation libraries (declarations for B&R ANSI C extensions) */
#include <bur/plctypes.h>

/**
Description:
    Library to converts base data types to an array of bytes, and an array of bytes to base data types as well as
    byte to an array of bits, and an array of bits to byte.

Note 1:
    A byte is a unit of storage in a computer which contains 8-bits and can store 256 different values: 0 to 255.

Note 2:
    BOOL (Bit)  : Boolean               [0, 1]          | 1-bit  | 0-Byte |
    USINT (Byte): Unsigned char         [0, 255]        | 8-bit  | 1-Byte |
    UINT        : Unsigned INT          [0, 65535]      | 16-bit | 2-Byte |
    UDINT       : Unsigned (double) INT [0, 4294967295] | 32-bit | 4-Byte |

Note 3:
    Bitwise Operators:
        &	Bitwise AND
        |	Bitwise OR
        <<	Shift left
        >>	Shift right
*/

typedef struct Convert_USINT_Array_To_UINT
{
	/**
	Description:
		Conversion of a vector of values (BYTES) to a value (UINT - 16-bit).
	*/

	/**
 	 * FUNCTION BLOCK: Convert_USINT_Array_To_UINT
	 * INPUT VARIABLES
 	 */
	USINT INPUT[2];

	/**
 	 * FUNCTION BLOCK: Convert_USINT_Array_To_UINT
	 * OUTPUT VARIABLES
 	 */
	UINT OUTPUT;
} Convert_USINT_Array_To_UINT_typ;

typedef struct Convert_USINT_Array_To_UDINT
{
	/**
	Description:
		Conversion of a vector of values (BYTES) to a value (UDINT - 32-bit).
	*/

	/**
 	 * FUNCTION BLOCK: Convert_USINT_Array_To_UDINT
	 * INPUT VARIABLES
 	 */
	USINT INPUT[4];

	/**
 	 * FUNCTION BLOCK: Convert_USINT_Array_To_UDINT
	 * OUTPUT VARIABLES
 	 */
	UDINT OUTPUT;
} Convert_USINT_Array_To_UDINT_typ;

typedef struct Convert_UINT_To_USINT_Array
{
	/**
	Description:
		Conversion of input value (UINT - 16-bit) into a vector of values (BYTES).
	*/

	/**
 	 * FUNCTION BLOCK: Convert_UINT_To_USINT_Array
	 * INPUT VARIABLES
 	 */
	UINT INPUT;

	/**
 	 * FUNCTION BLOCK: Convert_UINT_To_USINT_Array
	 * OUTPUT VARIABLES
 	 */
	USINT OUTPUT[2];
} Convert_UINT_To_USINT_Array_typ;

typedef struct Convert_UDINT_To_USINT_Array
{
	/**
	Description:
		Conversion of input value (UDINT - 32-bit) into a vector of values (BYTES).
	*/

	/**
 	 * FUNCTION BLOCK: Convert_UDINT_To_Byte_Array
	 * INPUT VARIABLES
 	 */
	UDINT INPUT;

	/**
 	 * FUNCTION BLOCK: Convert_UDINT_To_Byte_Array
	 * OUTPUT VARIABLES
 	 */
	USINT OUTPUT[4];
} Convert_UDINT_To_USINT_Array_typ;

typedef struct Convert_BOOL_Array_To_USINT
{
	/**
	Description:
		Conversion of input value (BYTE) into a vector of logical values (BITS = Booleans).
	*/

	/**
 	 * FUNCTION BLOCK: Convert_BOOL_Array_To_USINT
	 * INPUT VARIABLES
 	 */
	BOOL INPUT[8];

	/**
 	 * FUNCTION BLOCK: Convert_BOOL_Array_To_USINT
	 * OUTPUT VARIABLES
 	 */
	USINT OUTPUT;
} Convert_BOOL_Array_To_USINT_typ;

typedef struct Convert_USINT_To_BOOL_Array
{
	/**
	Description:
		Conversion of a vector of logical values (BITS = Booleans) to a value (BYTE).
	*/

	/**
 	 * FUNCTION BLOCK: Convert_USINT_To_BOOL_Array
	 * INPUT VARIABLES
 	 */
	USINT INPUT;

	/**
 	 * FUNCTION BLOCK: Convert_USINT_To_BOOL_Array
	 * OUTPUT VARIABLES
 	 */
	BOOL OUTPUT[8];
} Convert_USINT_To_BOOL_Array_typ;

/**
 * Declaration of function blocks for conversion between different types.
 */
_BUR_PUBLIC void Convert_USINT_Array_To_UINT(struct Convert_USINT_Array_To_UINT* inst);
_BUR_PUBLIC void Convert_USINT_Array_To_UDINT(struct Convert_USINT_Array_To_UDINT* inst);
_BUR_PUBLIC void Convert_UINT_To_USINT_Array(struct Convert_UINT_To_USINT_Array* inst);
_BUR_PUBLIC void Convert_UDINT_To_USINT_Array(struct Convert_UDINT_To_USINT_Array* inst);
_BUR_PUBLIC void Convert_BOOL_Array_To_USINT(struct Convert_BOOL_Array_To_USINT* inst);
_BUR_PUBLIC void Convert_USINT_To_BOOL_Array(struct Convert_USINT_To_BOOL_Array* inst);

void Convert_USINT_Array_To_UINT(struct Convert_USINT_Array_To_UINT* inst){
	/**
	Description:
		Conversion of a vector of values (BYTES) to a value (UINT - 16-bit).

	Args:
		(1) INPUT[0 .. 1] [BYTE (USINT) ARRAY]: Vector of values (BYTES).

	Returns:
		(1) OUTPUT [UINT]: A real number greater than or equal to zero.

	Example:
	     // Read inputs
		 inst->INPUT[0] = possible values range from 0 to 255
		 inst->INPUT[1] = possible values range from 0 to 255
		 // Call Function Block
		 Convert_USINT_Array_To_UINT(&inst);
		 // Write outputs
		 inst->OUTPUT = Result calculation from inst->IN_BYTE[0 .. 1] {possible values range from 0 to 65535}
	*/

	inst->OUTPUT = inst->INPUT[0] << 0x00 |
		inst->INPUT[1] << 0x08;
}

void Convert_USINT_Array_To_UDINT(struct Convert_USINT_Array_To_UDINT* inst){
	/**
	Description:
		Conversion of a vector of values (BYTES) to a value (UDINT - 32-bit).

	Args:
		(1) INPUT[0 .. 3] [BYTE (USINT) ARRAY]: Vector of values (BYTES).

	Returns:
		(1) OUTPUT [UDINT]: A real number greater than or equal to zero.

	Example:
	     // Read inputs
		 inst->INPUT[0] = possible values range from 0 to 255
		 ...
		 inst->INPUT[3] = possible values range from 0 to 255
		 // Call Function Block
		 Convert_USINT_Array_To_UDINT(&inst);
		 // Write outputs
		 inst->OUTPUT = Result calculation from inst->IN_BYTE[0 .. 3] {possible values range from 0 to 4294967295}
	*/

	inst->OUTPUT = inst->INPUT[0] << 0x00 |
		inst->INPUT[1] << 0x08 |
		inst->INPUT[2] << 0x10 |
		inst->INPUT[3] << 0x18;
}

void Convert_UINT_To_USINT_Array(struct Convert_UINT_To_USINT_Array* inst){
	/**
	Description:
		Conversion of input value (UINT - 16-bit) into a vector of values (BYTES).

	Args:
		(1) INPUT[UINT]: A real number greater than or equal to zero.

	Returns:
		(1) OUTPUT[0 .. 1] [BYTE (USINT) ARRAY]: Vector of values (BYTES).

	Example:
	     // Read inputs
		 inst->INPUT = possible values range from 0 to 65535
		 // Call Function Block
		 Convert_UINT_To_USINT_Array(&inst);
		 // Write outputs
		 inst->OUTPUT[0] = Result calculation from inst->IN_INT {Part 1: 0 .. 255}
		 inst->OUTPUT[1] = Result calculation from inst->IN_INT {Part 2: 0 .. 255}
	*/

	inst->OUTPUT[0] = (inst->INPUT >> 0x00) & 0xff;
	inst->OUTPUT[1] = (inst->INPUT >> 0x08) & 0xff;
}

void Convert_UDINT_To_USINT_Array(struct Convert_UDINT_To_USINT_Array* inst){
	/**
	Description:
		Conversion of input value (UDINT - 32-bit) into a vector of values (BYTES).

	Args:
		(1) INPUT [UDINT]: A real number greater than or equal to zero.

	Returns:
		(1) OUTPUT[0 .. 3] [BYTE (USINT) ARRAY]: Vector of values (BYTES).

	Example:
	     // Read inputs
		 inst->INPUT = possible values range from 0 to 4294967295
		 // Call Function Block
		 Convert_UDINT_To_USINT_Array(&inst);
		 // Write outputs
		 inst->OUTPUT[0] = Result calculation from inst->IN_UDINT {Part 1: 0 .. 255}
		 ...
		 inst->OUTPUT[3] = Result calculation from inst->IN_UDINT {Part 4: 0 .. 255}
	*/

	inst->OUTPUT[0] = (inst->INPUT >> 0x00) & 0xff;
	inst->OUTPUT[1] = (inst->INPUT >> 0x08) & 0xff;
	inst->OUTPUT[2] = (inst->INPUT >> 0x10) & 0xff;
	inst->OUTPUT[3] = (inst->INPUT >> 0x18) & 0xff;
}

void Convert_BOOL_Array_To_USINT(struct Convert_BOOL_Array_To_USINT* inst){
	/**
	Description:
		Conversion of input value (BYTE) into a vector of logical values (BITS = Booleans).

		Note:
			1 BYTE [0 - 255] = 8 BITs [0 - 1]

	Args:
		(1) INPUT[0 .. 7] [BIT (BOOL) ARRAY]: Vector of bits (1 BYTE).

	Returns:
		(1) OUTPUT [BYTE (USINT)]: A real number greater than or equal to zero.

	Example:
	     // Read inputs
		 inst->INPUT[0]  = possible values range from 0 (false) to 1 (true)
	     ...
		 inst->INPUT[7]  = possible values range from 0 (false) to 1 (true)
		 // Call Function Block
		 Convert_BOOL_Array_To_USINT(&inst);
		 // Write outputs
		 inst->OUTPUT = Result calculation from inst->IN_BIT[0 .. 7] {Part: 0 .. 255}
	*/

	inst->OUTPUT = inst->INPUT[0] << 0x00 |
		inst->INPUT[1] << 0x01 |
		inst->INPUT[2] << 0x02 |
		inst->INPUT[3] << 0x03 |
		inst->INPUT[4] << 0x04 |
		inst->INPUT[5] << 0x05 |
		inst->INPUT[6] << 0x06 |
		inst->INPUT[7] << 0x07;
}

void Convert_USINT_To_BOOL_Array(struct Convert_USINT_To_BOOL_Array* inst){
	/**
	Description:
		Conversion of a vector of logical values (BITS = Booleans) to a value (BYTE).

		Note:
			8 BITs [0 - 1] = 1 BYTE [0 - 255]

	Args:
		(1) INPUT [BYTE]: A real number greater than or equal to zero.

	Returns:
		(1) OUTPUT[0 .. 7] [BIT (BOOL) ARRAY]: Vector of bits (1 BYTE).

	Example:
	     // Read inputs
		 inst->INPUT  = possible values range from 0 to 255
		 // Call Function Block
		 Convert_USINT_To_BOOL_Array(&inst);
		 // Write outputs
		 inst->OUTPUT[0] = Result calculation from inst->IN_BYTE {Part 1: 0 (false) / 1 (true)}
		 ...
		 inst->OUTPUT[7] = Result calculation from inst->IN_BYTE {Part 1: 0 (false) / 1 (true)}
	*/

	inst->OUTPUT[0] = (inst->INPUT >> 0x00) & 0x01;
	inst->OUTPUT[1] = (inst->INPUT >> 0x01) & 0x01;
	inst->OUTPUT[2] = (inst->INPUT >> 0x02) & 0x01;
	inst->OUTPUT[3] = (inst->INPUT >> 0x03) & 0x01;
	inst->OUTPUT[4] = (inst->INPUT >> 0x04) & 0x01;
	inst->OUTPUT[5] = (inst->INPUT >> 0x05) & 0x01;
	inst->OUTPUT[6] = (inst->INPUT >> 0x06) & 0x01;
	inst->OUTPUT[7] = (inst->INPUT >> 0x07) & 0x01;
}

#endif
```

Listed in the project but not available here: Logical/T_ROB_2_L/Main.h, Logical/T_ROB_2_L/Converter.h, Logical/T_ROB_2_L/ABB_Library.h, Logical/T_ROB_2_L/Variables.var
